FUNCTION TryConvert_UINT_TO_REAL : BOOL
VAR_INPUT
	in : UINT;
	out : REFERENCE TO REAL;
END_VAR

out := UINT_TO_REAL(in);
TryConvert_UINT_TO_REAL := TRUE;

END_FUNCTION

(* stored: Version 1.1.0.1, ProductVersion 3.1.4024.12
   POU TryConvert_UINT_TO_REAL: Id {5af6f30b-ed68-4df6-9429-de2297a91fed}, SpecialFunc None *)
